// Mitsubishi GX Works2 project: Group3   PLC: FX3G

// global labels: Global1
VAR_GLOBAL
  start_day_x7 AT X007 : BOOL;
  break_working_m7 AT M7 : BOOL;
  label_working_y7 AT Y007 : BOOL;
  TC3_endDay AT TC3 : BOOL;
END_VAR
VAR_GLOBAL CONSTANT
  CONSTANT30_word : INT := 30;
END_VAR
VAR_GLOBAL
  TS3_endDay AT TS3 : BOOL;
  M_BLINKING_LIGHT1 AT M201 : BOOL;
  start_ziluf AT X010 : BOOL;
  M10_continueZiluf AT M10 : BOOL;
  stop_ziluf AT X005 : BOOL;
  sen_kremboIN AT X001 : BOOL;
  sen_kremboOUT AT X002 : BOOL;
  sen_30 AT X003 : BOOL;
  sen_15 AT X004 : BOOL;
  label_ziluf_working AT Y004 : BOOL;
  M0_help_blinking_light AT M0 : BOOL;
  TC0_timer_blinking AT TC0 : BOOL;
END_VAR
VAR_GLOBAL CONSTANT
  CONSTANT10_blinking : INT := 10;
END_VAR
VAR_GLOBAL
  TS0_output_timer_blinking AT TS0 : BOOL;
  TC1_timer_blinking AT TC1 : BOOL;
  TS1_output_timer_blinking AT TS1 : BOOL;
  M_BLINKING_LIGHT2 AT M202 : BOOL;
  RG_cream_input AT D1100 : REAL;
  RG_cream_container AT D1200 : REAL;
  RG_chocolate_input AT D1104 : REAL;
  RG_chocolate_container AT D1204 : REAL;
  RG_biskwit_input AT D1108 : REAL;
  RG_biskwit_container AT D1208 : REAL;
END_VAR
VAR_GLOBAL CONSTANT
  Cream_min_amount : REAL := 300;
END_VAR
VAR_GLOBAL
  M1_creamOK AT M1 : BOOL;
  M2_biskwitOK AT M2 : BOOL;
END_VAR
VAR_GLOBAL CONSTANT
  biskwit_min_amount : REAL := 6;
END_VAR
VAR_GLOBAL
  M3_chocolateOK AT M3 : BOOL;
END_VAR
VAR_GLOBAL CONSTANT
  Chocolate_two_dip_amount : REAL := 240;
END_VAR
VAR_GLOBAL
  cream_to_ziluf AT X011 : BOOL;
  RG_cream_ziluf AT D1300 : REAL;
END_VAR
VAR_GLOBAL CONSTANT
  CONSTANT_0 : REAL;
END_VAR
VAR_GLOBAL
  product_to_ziluf AT X011 : BOOL;
  M5_ziluf_stoped AT M5 : BOOL;
  M5_ziluf_can_start AT M5 : BOOL;
  not_ziluf_M11 AT M11 : BOOL;
  Move_to_chocolate AT M20 : BOOL;
  TC4_ziluf_chocolate AT TC4 : BOOL;
END_VAR
VAR_GLOBAL CONSTANT
  CONSTANT40_word : INT := 40;
END_VAR
VAR_GLOBAL
  TS4_end_ziluf_chocolate AT TS4 : BOOL;
  label_blink_ziluf_chocolate_y0 AT Y000 : BOOL;
  label_blink_ziluf_chocolate_y1 AT Y001 : BOOL;
  not_dip_M12 AT M12 : BOOL;
  RG_chocolate_dipping AT D1400 : REAL;
  sample_dip_type_x6 AT X006 : BOOL;
  M8_dipping_can_start AT M8 : BOOL;
  RG_Sample_dip_type AT D8280 : INT;
  RG_dip_value AT D1600 : INT;
END_VAR
VAR_GLOBAL CONSTANT
  CONSTANT400_word : INT := 400;
END_VAR
VAR_GLOBAL
  RG_dip_analog_value AT D1610 : INT;
END_VAR
VAR_GLOBAL CONSTANT
  CONSTANT5_word : INT := 5;
END_VAR
VAR_GLOBAL
  M91_one_dip AT M91 : BOOL;
END_VAR
VAR_GLOBAL CONSTANT
  Chocolate_one_dip_amount : REAL := 120;
  CONSTANT6_word : INT := 6;
END_VAR
VAR_GLOBAL
  M92_two_dip AT M92 : BOOL;
  M9_select_dip_type AT M9 : BOOL;
END_VAR
VAR_GLOBAL CONSTANT
  CONSTANT50_word : INT := 50;
END_VAR
VAR_GLOBAL
  TC5_diping_stage AT TC5 : BOOL;
  TS5_end_dipping_stage AT TS5 : BOOL;
  label_is_dipping_y3 AT Y003 : BOOL;
  pack_one_x0 AT X000 : BOOL;
  CC1_packing_stage AT CC1 : BOOL;
  CS1_last_packing AT CS1 : BOOL;
  label_alert_last_packing_y2 AT Y002 : BOOL;
  CC2_end_packing_stage AT CC2 : BOOL;
  CS2_end_packing AT CS2 : BOOL;
  TC6_diping_two_stage AT TC6 : BOOL;
  TS6_end_dipping_stage AT TS6 : BOOL;
  TC5_diping_one_stage AT TC5 : BOOL;
  RG_analog2_output AT D8282 : INT;
  RG_finished_daily_krembos AT D1700 : REAL;
END_VAR
VAR_GLOBAL CONSTANT
  CONSTANT10_word : INT := 10;
END_VAR
VAR_GLOBAL
  M95_end_packing AT M95 : BOOL;
END_VAR
VAR_GLOBAL CONSTANT
  CONSTANT400_float : REAL := 400;
END_VAR
VAR_GLOBAL
  RG_finished_krembos_float AT D1710 : REAL;
END_VAR
VAR_GLOBAL CONSTANT
  CONSTANT6_float : REAL := 6;
  CONSTANT40_float : REAL := 40;
END_VAR
VAR_GLOBAL
  not_pack_M13 AT M13 : BOOL;
END_VAR
VAR_GLOBAL CONSTANT
  CONSTANT_0_WORD : INT;
END_VAR

// task Task_01 (event TRUE, interval 0, priority 31): POU_01

PROGRAM POU_01
(* structured ladder/FBD written out as ST: instructions are called as NAME(EN, inputs, outputs); _pN, _eN, _tN stand for wires *)
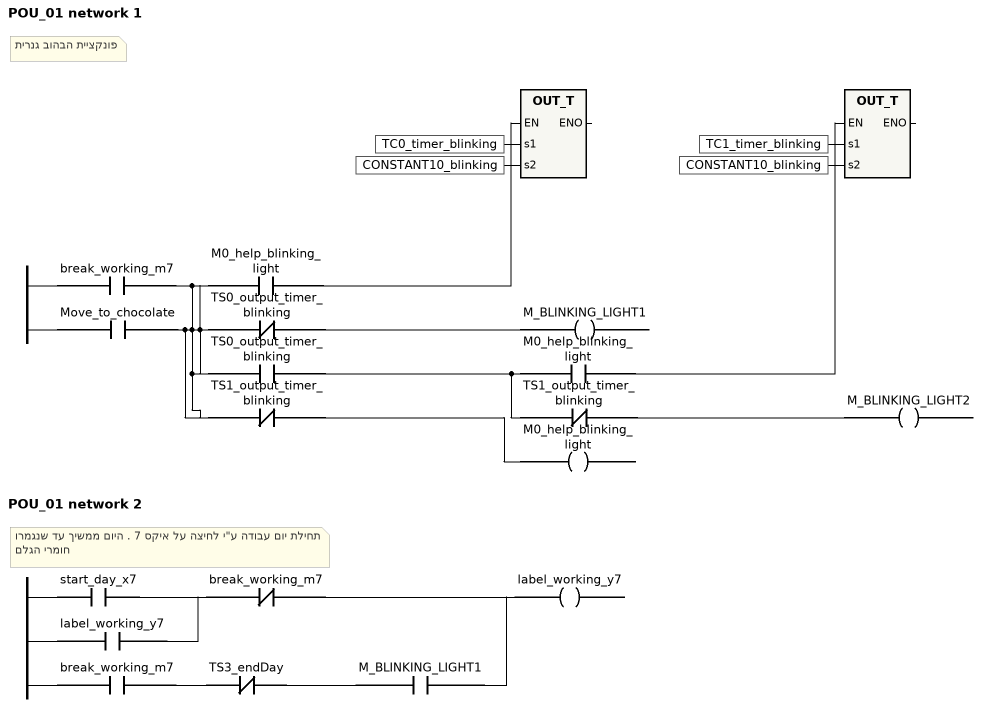
(* network 1 *)
(* פונקציית הבהוב גנרית *)
_p1 := break_working_m7 OR Move_to_chocolate;
OUT_T(_p1 AND M0_help_blinking_light, TC0_timer_blinking, CONSTANT10_blinking);
M_BLINKING_LIGHT1 := _p1 AND NOT TS0_output_timer_blinking;
_p2 := _p1 AND TS0_output_timer_blinking;
OUT_T(_p2 AND M0_help_blinking_light, TC1_timer_blinking, CONSTANT10_blinking);
M_BLINKING_LIGHT2 := _p2 AND NOT TS1_output_timer_blinking;
M0_help_blinking_light := _p1 AND NOT TS1_output_timer_blinking;
(* network 2 *)
(* תחילת יום עבודה ע"י לחיצה על איקס 7 . היום ממשיך עד שנגמרו חומרי הגלם *)
label_working_y7 := ((start_day_x7 OR label_working_y7) AND NOT break_working_m7) OR (break_working_m7 AND NOT TS3_endDay AND M_BLINKING_LIGHT1);
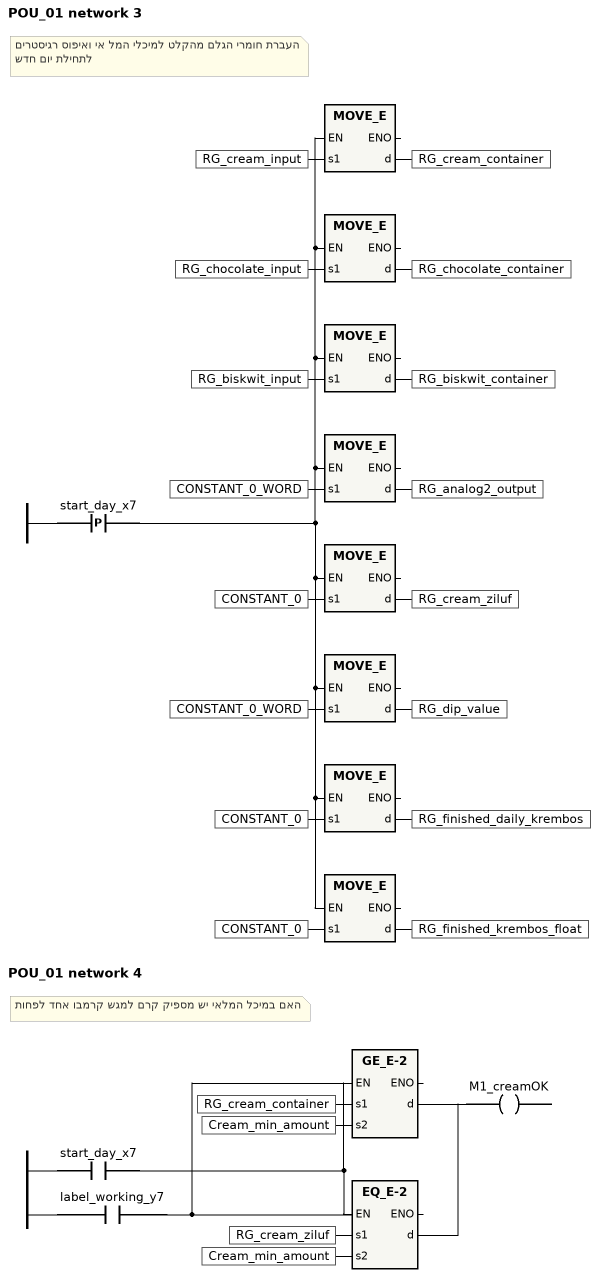
(* network 3 *)
(* העברת חומרי הגלם מהקלט למיכלי המל אי ואיפוס רגיסטרים לתחילת יום חדש *)
_p1 := LDP(TRUE, start_day_x7);
MOVE_E(_p1, RG_cream_input, RG_cream_container);
MOVE_E(_p1, RG_chocolate_input, RG_chocolate_container);
MOVE_E(_p1, RG_biskwit_input, RG_biskwit_container);
MOVE_E(_p1, CONSTANT_0_WORD, RG_analog2_output);
MOVE_E(_p1, CONSTANT_0, RG_cream_ziluf);
MOVE_E(_p1, CONSTANT_0_WORD, RG_dip_value);
MOVE_E(_p1, CONSTANT_0, RG_finished_daily_krembos);
MOVE_E(_p1, CONSTANT_0, RG_finished_krembos_float);
(* network 4 *)
(* האם במיכל המלאי יש מספיק קרם למגש קרמבו אחד לפחות *)
_p1 := start_day_x7 OR label_working_y7;
GE_E(_p1, RG_cream_container, Cream_min_amount, _t2);
EQ_E(_p1, RG_cream_ziluf, Cream_min_amount, _t3);
M1_creamOK := _t2 OR _t3;
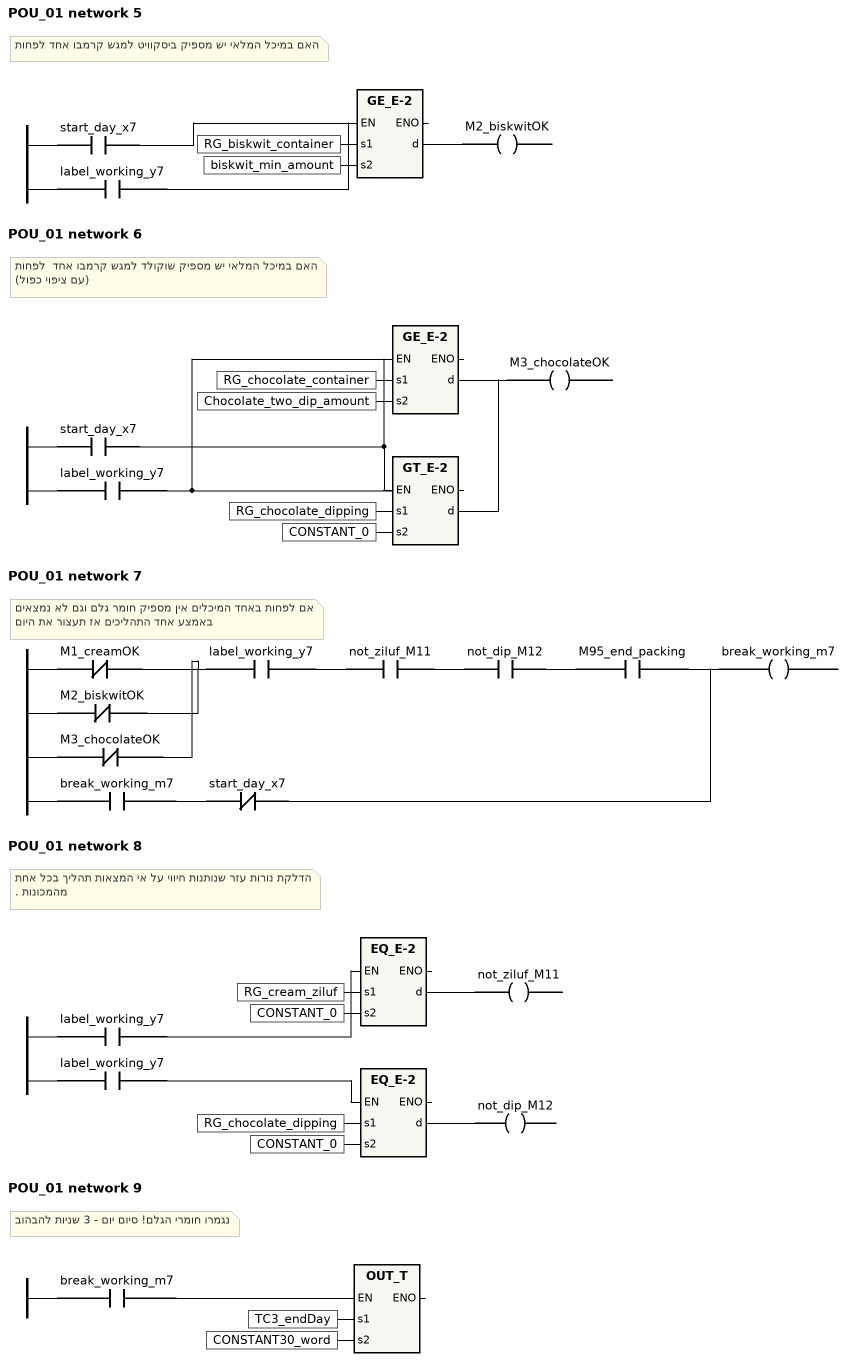
(* network 5 *)
(* האם במיכל המלאי יש מספיק ביסקוויט למגש קרמבו אחד לפחות *)
GE_E(start_day_x7 OR label_working_y7, RG_biskwit_container, biskwit_min_amount, _t1);
M2_biskwitOK := _t1;
(* network 6 *)
(* האם במיכל המלאי יש מספיק שוקולד למגש קרמבו אחד  לפחות (עם ציפוי כפול) *)
_p1 := start_day_x7 OR label_working_y7;
GE_E(_p1, RG_chocolate_container, Chocolate_two_dip_amount, _t2);
GT_E(_p1, RG_chocolate_dipping, CONSTANT_0, _t3);
M3_chocolateOK := _t2 OR _t3;
(* network 7 *)
(* אם לפחות באחד המיכלים אין מספיק חומר גלם וגם לא נמצאים באמצע אחד התהליכים אז תעצור את היום *)
break_working_m7 := ((((((NOT M1_creamOK) OR (NOT M2_biskwitOK) OR (NOT M3_chocolateOK)) AND label_working_y7) AND not_ziluf_M11) AND not_dip_M12) AND M95_end_packing) OR (break_working_m7 AND NOT start_day_x7);
(* network 8 *)
(* הדלקת נורות עזר שנותנות חיווי על אי המצאות תהליך בכל אחת מהמכונות . *)
EQ_E(label_working_y7, RG_cream_ziluf, CONSTANT_0, _t1);
not_ziluf_M11 := _t1;
EQ_E(label_working_y7, RG_chocolate_dipping, CONSTANT_0, _t2);
not_dip_M12 := _t2;
(* network 9 *)
(* נגמרו חומרי הגלם! סיום יום - 3 שניות להבהוב *)
OUT_T(break_working_m7, TC3_endDay, CONSTANT30_word);
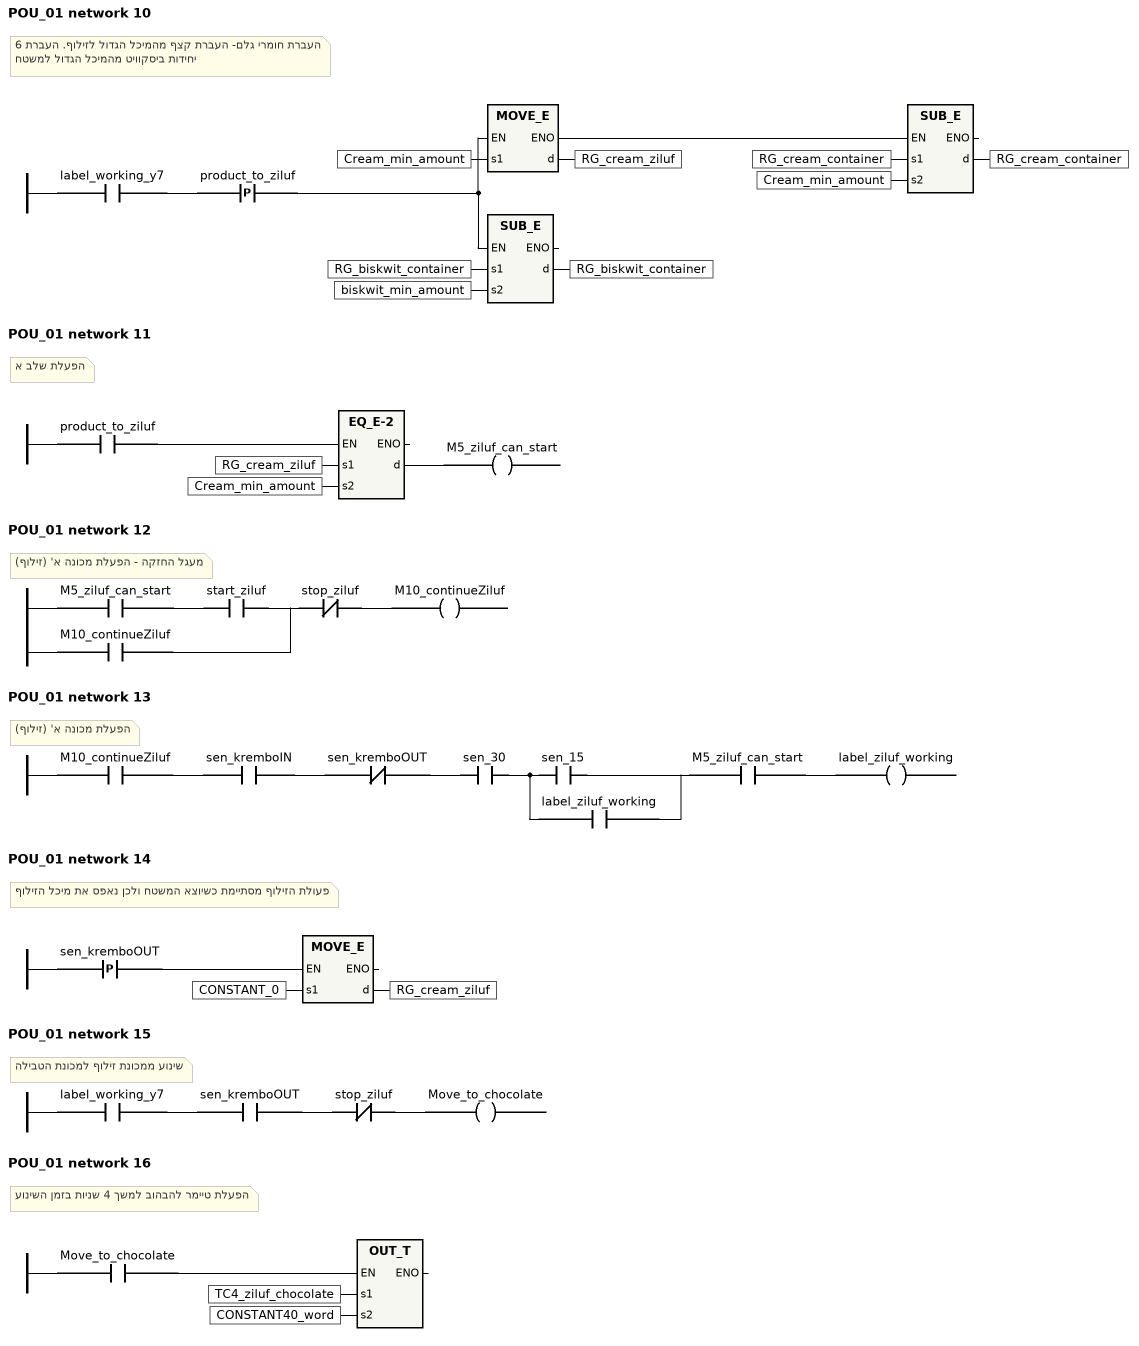
(* network 10 *)
(* העברת חומרי גלם- העברת קצף מהמיכל הגדול לזילוף. העברת 6 יחידות ביסקוויט מהמיכל הגדול למשטח *)
_p1 := label_working_y7 AND LDP(TRUE, product_to_ziluf);
_e2 := MOVE_E(_p1, Cream_min_amount, RG_cream_ziluf);
SUB_E(_e2, RG_cream_container, Cream_min_amount, RG_cream_container);
SUB_E(_p1, RG_biskwit_container, biskwit_min_amount, RG_biskwit_container);
(* network 11 *)
(* הפעלת שלב א *)
EQ_E(product_to_ziluf, RG_cream_ziluf, Cream_min_amount, _t1);
M5_ziluf_can_start := _t1;
(* network 12 *)
(* מעגל החזקה - הפעלת מכונה א' (זילוף) *)
M10_continueZiluf := ((M5_ziluf_can_start AND start_ziluf) OR M10_continueZiluf) AND NOT stop_ziluf;
(* network 13 *)
(* הפעלת מכונה א' (זילוף) *)
_p1 := M10_continueZiluf AND sen_kremboIN AND NOT sen_kremboOUT AND sen_30;
label_ziluf_working := ((_p1 AND sen_15) OR (_p1 AND label_ziluf_working)) AND M5_ziluf_can_start;
(* network 14 *)
(* פעולת הזילוף מסתיימת כשיוצא המשטח ולכן נאפס את מיכל הזילוף *)
MOVE_E(LDP(TRUE, sen_kremboOUT), CONSTANT_0, RG_cream_ziluf);
(* network 15 *)
(* שינוע ממכונת זילוף למכונת הטבילה *)
Move_to_chocolate := label_working_y7 AND sen_kremboOUT AND NOT stop_ziluf;
(* network 16 *)
(* הפעלת טיימר להבהוב למשך 4 שניות בזמן השינוע *)
OUT_T(Move_to_chocolate, TC4_ziluf_chocolate, CONSTANT40_word);
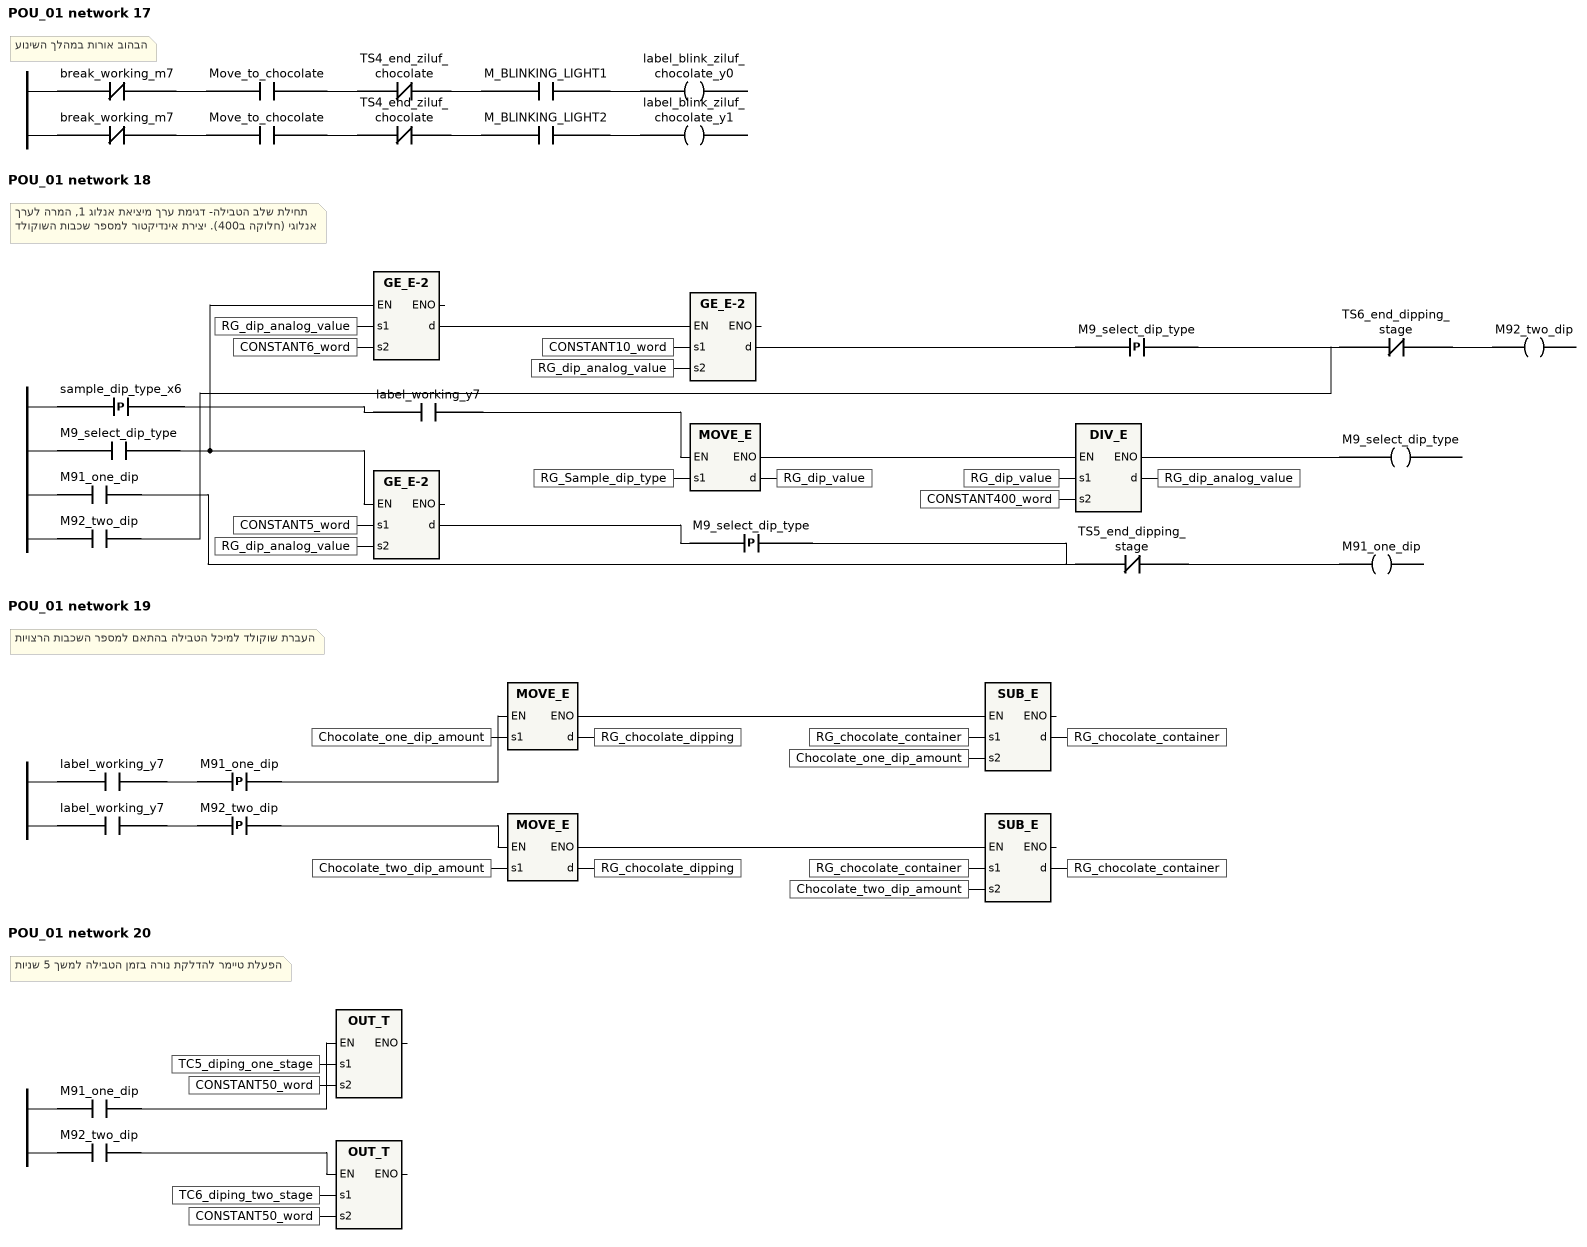
(* network 17 *)
(* הבהוב אורות במהלך השינוע *)
label_blink_ziluf_chocolate_y0 := NOT break_working_m7 AND Move_to_chocolate AND NOT TS4_end_ziluf_chocolate AND M_BLINKING_LIGHT1;
label_blink_ziluf_chocolate_y1 := NOT break_working_m7 AND Move_to_chocolate AND NOT TS4_end_ziluf_chocolate AND M_BLINKING_LIGHT2;
(* network 18 *)
(* תחילת שלב הטבילה- דגימת ערך מיציאת אנלוג 1, המרה לערך אנלוגי (חלוקה ב400). יצירת אינדיקטור למספר שכבות השוקולד *)
_e1 := MOVE_E(LDP(TRUE, sample_dip_type_x6) AND label_working_y7, RG_Sample_dip_type, RG_dip_value);
_e2 := DIV_E(_e1, RG_dip_value, CONSTANT400_word, RG_dip_analog_value);
M9_select_dip_type := _e2;
GE_E(M9_select_dip_type, CONSTANT5_word, RG_dip_analog_value, _t3);
M91_one_dip := ((_t3 AND LDP(TRUE, M9_select_dip_type)) OR M91_one_dip) AND NOT TS5_end_dipping_stage;
GE_E(M9_select_dip_type, RG_dip_analog_value, CONSTANT6_word, _t4);
GE_E(_t4, CONSTANT10_word, RG_dip_analog_value, _t5);
M92_two_dip := ((_t5 AND LDP(TRUE, M9_select_dip_type)) OR M92_two_dip) AND NOT TS6_end_dipping_stage;
(* network 19 *)
(* העברת שוקולד למיכל הטבילה בהתאם למספר השכבות הרצויות *)
_e1 := MOVE_E(label_working_y7 AND LDP(TRUE, M91_one_dip), Chocolate_one_dip_amount, RG_chocolate_dipping);
SUB_E(_e1, RG_chocolate_container, Chocolate_one_dip_amount, RG_chocolate_container);
_e2 := MOVE_E(label_working_y7 AND LDP(TRUE, M92_two_dip), Chocolate_two_dip_amount, RG_chocolate_dipping);
SUB_E(_e2, RG_chocolate_container, Chocolate_two_dip_amount, RG_chocolate_container);
(* network 20 *)
(* הפעלת טיימר להדלקת נורה בזמן הטבילה למשך 5 שניות *)
OUT_T(M91_one_dip, TC5_diping_one_stage, CONSTANT50_word);
OUT_T(M92_two_dip, TC6_diping_two_stage, CONSTANT50_word);
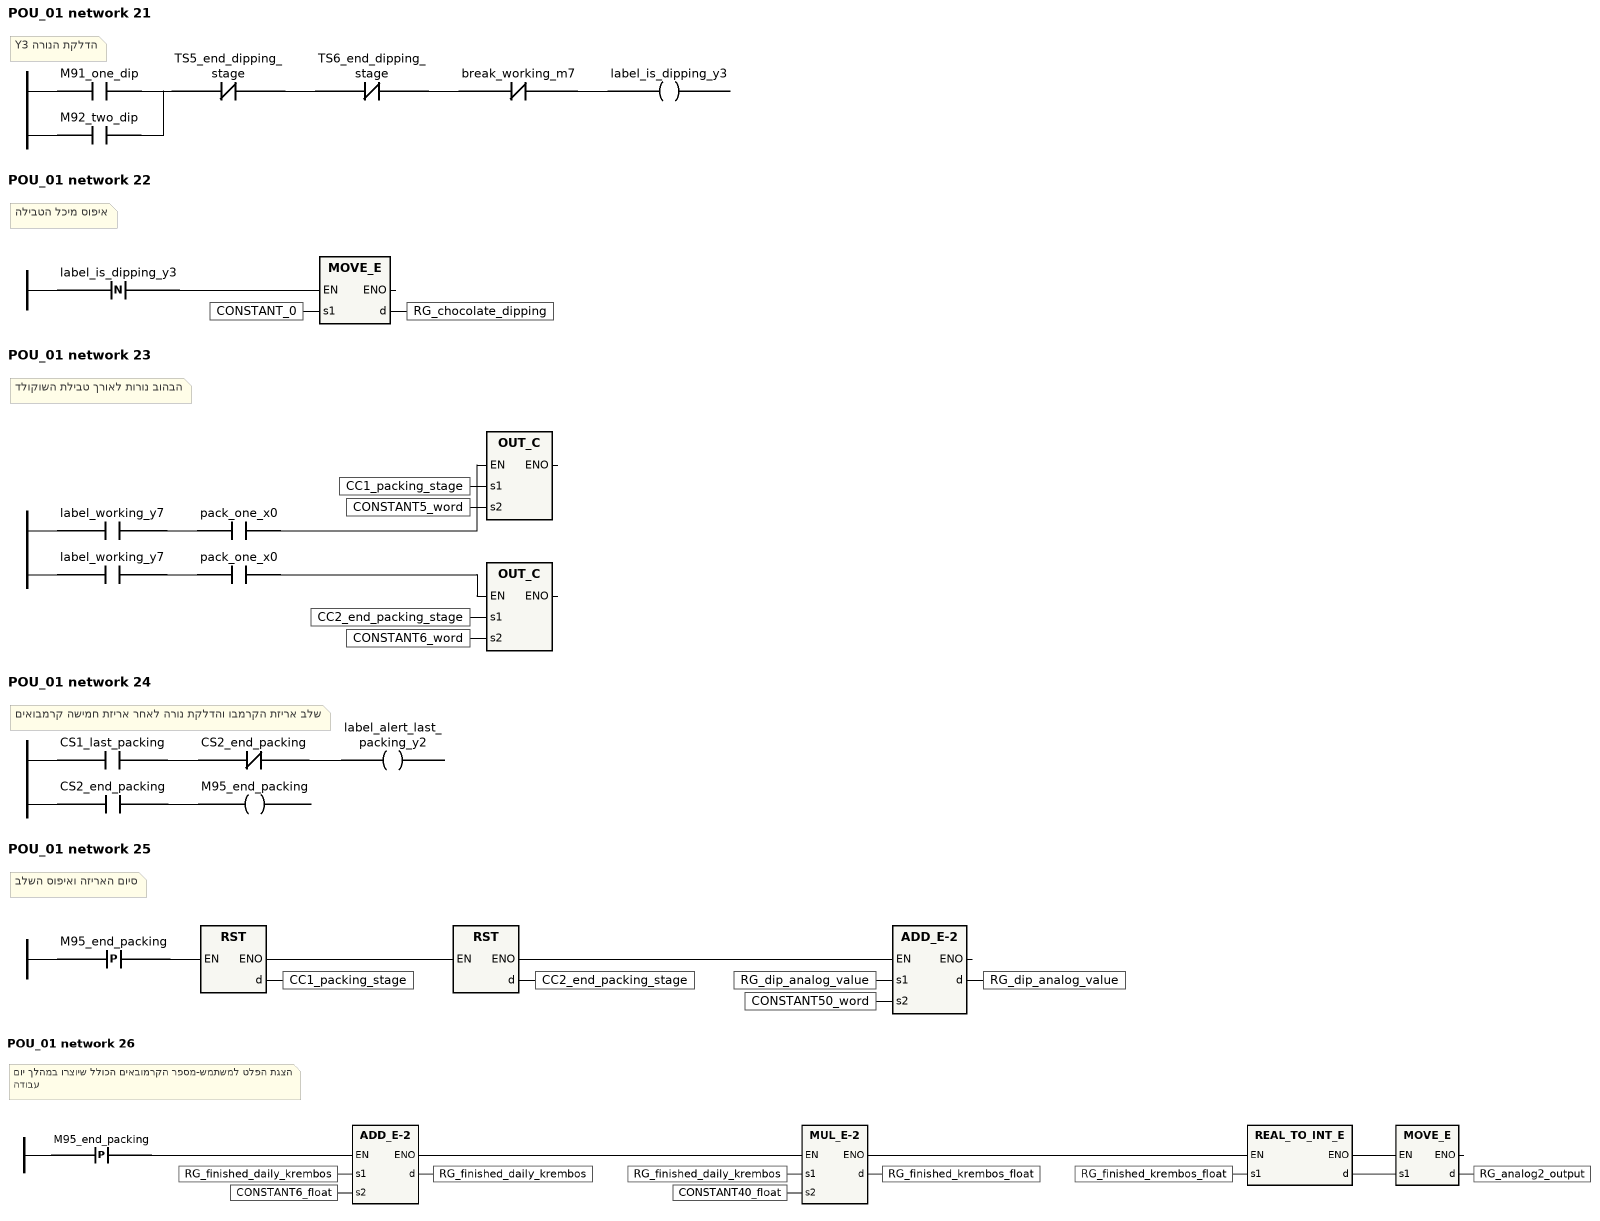
(* network 21 *)
(* הדלקת הנורה Y3 *)
label_is_dipping_y3 := (((M91_one_dip OR M92_two_dip) AND NOT TS5_end_dipping_stage) AND NOT TS6_end_dipping_stage) AND NOT break_working_m7;
(* network 22 *)
(* איפוס מיכל הטבילה *)
MOVE_E(LDF(TRUE, label_is_dipping_y3), CONSTANT_0, RG_chocolate_dipping);
(* network 23 *)
(* הבהוב נורות לאורך טבילת השוקולד *)
OUT_C(label_working_y7 AND pack_one_x0, CC1_packing_stage, CONSTANT5_word);
OUT_C(label_working_y7 AND pack_one_x0, CC2_end_packing_stage, CONSTANT6_word);
(* network 24 *)
(* שלב אריזת הקרמבו והדלקת נורה לאחר אריזת חמישה קרמבואים *)
label_alert_last_packing_y2 := CS1_last_packing AND NOT CS2_end_packing;
M95_end_packing := CS2_end_packing;
(* network 25 *)
(* סיום האריזה ואיפוס השלב *)
_e1 := RST(LDP(TRUE, M95_end_packing), CC1_packing_stage);
_e2 := RST(_e1, CC2_end_packing_stage);
ADD_E(_e2, RG_dip_analog_value, CONSTANT50_word, RG_dip_analog_value);
(* network 26 *)
(* הצגת הפלט למשתמש-מספר הקרמובאים הכולל שיוצרו במהלך יום עבודה *)
_e1 := ADD_E(LDP(TRUE, M95_end_packing), RG_finished_daily_krembos, CONSTANT6_float, RG_finished_daily_krembos);
_e2 := MUL_E(_e1, RG_finished_daily_krembos, CONSTANT40_float, RG_finished_krembos_float);
_e4 := REAL_TO_INT_E(_e2, RG_finished_krembos_float, _t3);
MOVE_E(_e4, _t3, RG_analog2_output);
END_PROGRAM
